(* PLC project motor_driver, Unknown motor_driver 1 *)
(* stored: creationDateTime 2024-07-05T11:44:58, modificationDateTime 2024-07-08T09:22:17 *)

FUNCTION GET_ON_TIME : TIME
  VAR_INPUT
    duty_cycle : UINT;
  END_VAR
  VAR
    local_time : TIME;
  END_VAR

            IF (duty_cycle = 0) THEN

  GET_ON_TIME := T#0ms;

  RETURN;



ELSIF duty_cycle = 1 THEN

  GET_ON_TIME := T#0.02ms;

	RETURN;

  

ELSIF duty_cycle = 2 THEN

  GET_ON_TIME := T#0.04ms;

  RETURN;

  

ELSIF duty_cycle = 3 THEN

  GET_ON_TIME := T#0.06ms;

  RETURN;

  

ELSIF duty_cycle = 4 THEN

  GET_ON_TIME := T#0.08ms;

  RETURN;

  

ELSIF duty_cycle = 5 THEN

  GET_ON_TIME := T#0.1ms;

  RETURN;

  

ELSIF duty_cycle = 6 THEN

  GET_ON_TIME := T#0.12ms;

  RETURN;



ELSIF duty_cycle = 7 THEN

  GET_ON_TIME := T#0.14ms;

  RETURN;

  

ELSIF duty_cycle = 8 THEN

  GET_ON_TIME := T#0.16ms;

  RETURN;

    

ELSIF duty_cycle = 9 THEN

  GET_ON_TIME := T#0.18ms;

  RETURN;

  

ELSIF duty_cycle = 10 THEN

  GET_ON_TIME := T#0.2ms;

  RETURN;



ELSIF duty_cycle = 11 THEN

  GET_ON_TIME := T#0.22ms;

  RETURN;



ELSIF duty_cycle = 12 THEN

  GET_ON_TIME := T#0.24ms;

  RETURN;



ELSIF duty_cycle = 13 THEN

  GET_ON_TIME := T#0.26ms;

  RETURN;



ELSIF duty_cycle = 14 THEN

  GET_ON_TIME := T#0.28ms;

  RETURN;



ELSIF duty_cycle = 15 THEN

  GET_ON_TIME := T#0.3ms;

  RETURN;



ELSIF duty_cycle = 16 THEN

  GET_ON_TIME := T#0.32ms;

  RETURN;



ELSIF duty_cycle = 17 THEN

  GET_ON_TIME := T#0.34ms;

  RETURN;



ELSIF duty_cycle = 18 THEN

  GET_ON_TIME := T#0.36ms;

  RETURN;



ELSIF duty_cycle = 19 THEN

  GET_ON_TIME := T#0.38ms;

  RETURN;



ELSIF duty_cycle = 20 THEN

  GET_ON_TIME := T#0.4ms;

  RETURN;



ELSIF duty_cycle = 21 THEN

  GET_ON_TIME := T#0.42ms;

  RETURN;



ELSIF duty_cycle = 22 THEN

  GET_ON_TIME := T#0.44ms;

  RETURN;



ELSIF duty_cycle = 23 THEN

  GET_ON_TIME := T#0.46ms;

  RETURN;



ELSIF duty_cycle = 24 THEN

  GET_ON_TIME := T#0.48ms;

  RETURN;



ELSIF duty_cycle = 25 THEN

  GET_ON_TIME := T#0.5ms;

  RETURN;



ELSIF duty_cycle = 26 THEN

  GET_ON_TIME := T#0.52ms;

  RETURN;



ELSIF duty_cycle = 27 THEN

  GET_ON_TIME := T#0.54ms;

  RETURN;



ELSIF duty_cycle = 28 THEN

  GET_ON_TIME := T#0.56ms;

  RETURN;



ELSIF duty_cycle = 29 THEN

  GET_ON_TIME := T#0.58ms;

  RETURN;



ELSIF duty_cycle = 30 THEN

  GET_ON_TIME := T#0.6ms;

  RETURN;



ELSIF duty_cycle = 31 THEN

  GET_ON_TIME := T#0.62ms;

  RETURN;



ELSIF duty_cycle = 32 THEN

  GET_ON_TIME := T#0.64ms;

  RETURN;



ELSIF duty_cycle = 33 THEN

  GET_ON_TIME := T#0.66ms;

  RETURN;



ELSIF duty_cycle = 34 THEN

  GET_ON_TIME := T#0.68ms;

  RETURN;



ELSIF duty_cycle = 35 THEN

  GET_ON_TIME := T#0.7ms;

  RETURN;



ELSIF duty_cycle = 36 THEN

  GET_ON_TIME := T#0.72ms;

  RETURN;



ELSIF duty_cycle = 37 THEN

  GET_ON_TIME := T#0.74ms;

  RETURN;



ELSIF duty_cycle = 38 THEN

  GET_ON_TIME := T#0.76ms;

  RETURN;



ELSIF duty_cycle = 39 THEN

  GET_ON_TIME := T#0.78ms;

  RETURN;



ELSIF duty_cycle = 40 THEN

  GET_ON_TIME := T#0.8ms;

  RETURN;



ELSIF duty_cycle = 41 THEN

  GET_ON_TIME := T#0.82ms;

  RETURN;



ELSIF duty_cycle = 42 THEN

  GET_ON_TIME := T#0.84ms;

  RETURN;



ELSIF duty_cycle = 43 THEN

  GET_ON_TIME := T#0.86ms;

  RETURN;



ELSIF duty_cycle = 44 THEN

  GET_ON_TIME := T#0.88ms;

  RETURN;



ELSIF duty_cycle = 45 THEN

  GET_ON_TIME := T#0.9ms;

  RETURN;



ELSIF duty_cycle = 46 THEN

  GET_ON_TIME := T#0.92ms;

  RETURN;



ELSIF duty_cycle = 47 THEN

  GET_ON_TIME := T#0.94ms;

  RETURN;



ELSIF duty_cycle = 48 THEN

  GET_ON_TIME := T#0.96ms;

  RETURN;



ELSIF duty_cycle = 49 THEN

  GET_ON_TIME := T#0.98ms;

  RETURN;



ELSIF duty_cycle = 50 THEN

  GET_ON_TIME := T#1ms;

  RETURN;



ELSIF duty_cycle = 51 THEN

  GET_ON_TIME := T#1.02ms;

  RETURN;



ELSIF duty_cycle = 52 THEN

  GET_ON_TIME := T#1.04ms;

  RETURN;



ELSIF duty_cycle = 53 THEN

  GET_ON_TIME := T#1.06ms;

  RETURN;



ELSIF duty_cycle = 54 THEN

  GET_ON_TIME := T#1.08ms;

  RETURN;



ELSIF duty_cycle = 55 THEN

  GET_ON_TIME := T#1.1ms;

  RETURN;



ELSIF duty_cycle = 56 THEN

  GET_ON_TIME := T#1.12ms;

  RETURN;



ELSIF duty_cycle = 57 THEN

  GET_ON_TIME := T#1.14ms;

  RETURN;

  

ELSIF duty_cycle = 58 THEN

  GET_ON_TIME := T#1.16ms;

  RETURN;



ELSIF duty_cycle = 59 THEN

  GET_ON_TIME := T#1.18ms;

  RETURN;



ELSIF duty_cycle = 60 THEN

  GET_ON_TIME := T#1.2ms;

  RETURN;



ELSIF duty_cycle = 61 THEN

  GET_ON_TIME := T#1.22ms;

  RETURN;



ELSIF duty_cycle = 62 THEN

  GET_ON_TIME := T#1.24ms;

  RETURN;



ELSIF duty_cycle = 63 THEN

  GET_ON_TIME := T#1.26ms;

  RETURN;



ELSIF duty_cycle = 64 THEN

  GET_ON_TIME := T#1.28ms;

  RETURN;



ELSIF duty_cycle = 65 THEN

  GET_ON_TIME := T#1.3ms;

  RETURN;



ELSIF duty_cycle = 66 THEN

  GET_ON_TIME := T#1.32ms;

  RETURN;



ELSIF duty_cycle = 67 THEN

  GET_ON_TIME := T#1.34ms;

  RETURN;



ELSIF duty_cycle = 68 THEN

  GET_ON_TIME := T#1.36ms;

  RETURN;



ELSIF duty_cycle = 69 THEN

  GET_ON_TIME := T#1.38ms;

  RETURN;



ELSIF duty_cycle = 70 THEN

  GET_ON_TIME := T#1.4ms;

  RETURN;



ELSIF duty_cycle = 71 THEN

  GET_ON_TIME := T#1.42ms;

  RETURN;



ELSIF duty_cycle = 72 THEN

  GET_ON_TIME := T#1.44ms;

  RETURN;



ELSIF duty_cycle = 73 THEN

  GET_ON_TIME := T#1.46ms;

  RETURN;



ELSIF duty_cycle = 74 THEN

  GET_ON_TIME := T#1.48ms;

  RETURN;



ELSIF duty_cycle = 75 THEN

  GET_ON_TIME := T#1.5ms;

  RETURN;



ELSIF duty_cycle = 76 THEN

  GET_ON_TIME := T#1.52ms;

  RETURN;



ELSIF duty_cycle = 77 THEN

  GET_ON_TIME := T#1.54ms;

  RETURN;



ELSIF duty_cycle = 78 THEN

  GET_ON_TIME := T#1.56ms;

  RETURN;



ELSIF duty_cycle = 79 THEN

  GET_ON_TIME := T#1.58ms;

  RETURN;



ELSIF duty_cycle = 80 THEN

  GET_ON_TIME := T#1.6ms;

  RETURN;



ELSIF duty_cycle = 81 THEN

  GET_ON_TIME := T#1.62ms;

  RETURN;



ELSIF duty_cycle = 82 THEN

  GET_ON_TIME := T#1.64ms;

  RETURN;



ELSIF duty_cycle = 83 THEN

  GET_ON_TIME := T#1.66ms;

  RETURN;



ELSIF duty_cycle = 84 THEN

  GET_ON_TIME := T#1.68ms;

  RETURN;



ELSIF duty_cycle = 85 THEN

  GET_ON_TIME := T#1.7ms;

  RETURN;



ELSIF duty_cycle = 86 THEN

  GET_ON_TIME := T#1.72ms;

  RETURN;



ELSIF duty_cycle = 87 THEN

  GET_ON_TIME := T#1.74ms;

  RETURN;

  

ELSIF duty_cycle = 88 THEN

  GET_ON_TIME := T#1.76ms;

  RETURN;



ELSIF duty_cycle = 89 THEN

  GET_ON_TIME := T#1.78ms;

  RETURN;



ELSIF duty_cycle = 90 THEN

  GET_ON_TIME := T#1.8ms;

  RETURN;

  

ELSIF duty_cycle = 91 THEN

  GET_ON_TIME := T#1.82ms;

  RETURN;



ELSIF duty_cycle = 92 THEN

  GET_ON_TIME := T#1.84ms;

  RETURN;



ELSIF duty_cycle = 93 THEN

  GET_ON_TIME := T#1.86ms;

  RETURN;



ELSIF duty_cycle = 94 THEN

  GET_ON_TIME := T#1.88ms;

  RETURN;



ELSIF duty_cycle = 95 THEN

  GET_ON_TIME := T#1.9ms;

  RETURN;



ELSIF duty_cycle = 96 THEN

  GET_ON_TIME := T#1.92ms;

  RETURN;



ELSIF duty_cycle = 97 THEN

  GET_ON_TIME := T#1.94ms;

  RETURN;



ELSIF duty_cycle = 98 THEN

  GET_ON_TIME := T#1.96ms;

  RETURN;



ELSIF duty_cycle = 99 THEN

  GET_ON_TIME := T#1.98ms;

  RETURN;



ELSIF duty_cycle = 100 THEN

  GET_ON_TIME := T#2ms;

  RETURN;



END_IF;


          
END_FUNCTION

PROGRAM motor_driver
  VAR
    led AT %QX0.3 : BOOL;
  END_VAR
  VAR
    output_on_timer : TON;
    output_off_timer : TOF;
    input_angle : INT := 90;
    real_angle : REAL := 90.0;
    duty_cycle : UINT := 50;
    on_PT : TIME := T#1ms;
    off_PT : TIME := T#1ms;
  END_VAR
  VAR
    output_pin AT %QW1 : UINT := 65535;
  END_VAR

            (* validate the servo angle *)
IF(input_angle < 0) THEN
  input_angle := 0;

ELSIF(input_angle > 180) THEN
  input_angle := 180;

END_IF;

(* control the servo *)
real_angle := INT_TO_REAL(input_angle);
duty_cycle := REAL_TO_UINT(100.0 / 180.0 * real_angle);

on_PT := GET_ON_TIME(duty_cycle);

output_on_timer(IN := NOT(output_off_timer.Q), PT := on_PT);
output_off_timer(IN := output_on_timer.Q, PT := off_PT);

IF output_on_timer.Q THEN
  output_pin := 65535;
  
ELSE
  output_pin := 0;

END_IF;

(* Blink the builtin LED *)
led := output_on_timer.Q;

          
END_PROGRAM

CONFIGURATION Config0
  RESOURCE Res0 ON PLC
    TASK task0(INTERVAL := T#2ms, PRIORITY := 0);
    PROGRAM instance0 WITH task0 : motor_driver;
  END_RESOURCE
END_CONFIGURATION
